PROGRAM GetLocalPlcEx
VAR
	fbPLCDBRead : FB_PLCDBReadEvt (sNetID := '', tTimeout := T#5S);
	ColumnNames_read : ARRAY [0..4] OF STRING(50);
	myDBID: uint := 1;
	sMyTableName : T_MaxString:='Data';
	myRecordRead : stData;
	tcMessage_read : I_TcMessage;

	fbTon: TON;
	bRead: bool;
END_VAR

fbTon(IN:= NOT fbTon.Q, PT:= T#200MS);
IF fbTon.Q THEN
	bRead:= TRUE;
END_IF

IF bRead THEN
	ColumnNames_read[0] := 'ID';
	ColumnNames_read[1] := 'Timestamp';
	ColumnNames_read[2] := 'Speed';
	ColumnNames_read[3] := 'Pos';
	ColumnNames_read[4] := 'Pulse';
	
	IF fbPLCDBRead.ReadStruct(
		hDBID:= myDBID,
		sTableName:= sMyTableName,
		pColumnNames:= ADR(ColumnNames_read),
		cbColumnNames:= SIZEOF(ColumnNames_read),
		sOrderByColumn:= 'ID', 
		eOrderType:= E_OrderType.DESC, 
		nStartIndex:= 0, 
		nRecordCount:= 1, 
		pData:= ADR(myRecordRead), 
		cbData:= SIZEOF(myRecordRead)
	)
	THEN
		IF fbPLCDBRead.bError THEN
		tcMessage_read := fbPLCDBRead.ipTcResult;
		END_IF
		bRead:= FALSE;
	END_IF	
END_IF

END_PROGRAM

(* stored: Version 1.1.0.1, ProductVersion 3.1.4024.4
   POU GetLocalPlcEx: Id {c4b72cc0-13bc-4bc0-a837-24944c1ee986}, SpecialFunc None *)
